# EPICS autosave request: GALILMUL/iocBoot/iocGALILMUL-IOC-01/GALILMUL_01_settings.req
file "GALIL_controller_settings.req" "P=$(P),CCP=$(MTRCTRL1)"
file "GALIL_controller_settings.req" "P=$(P),CCP=$(MTRCTRL2)"
